RoboDK station: V1.rdk

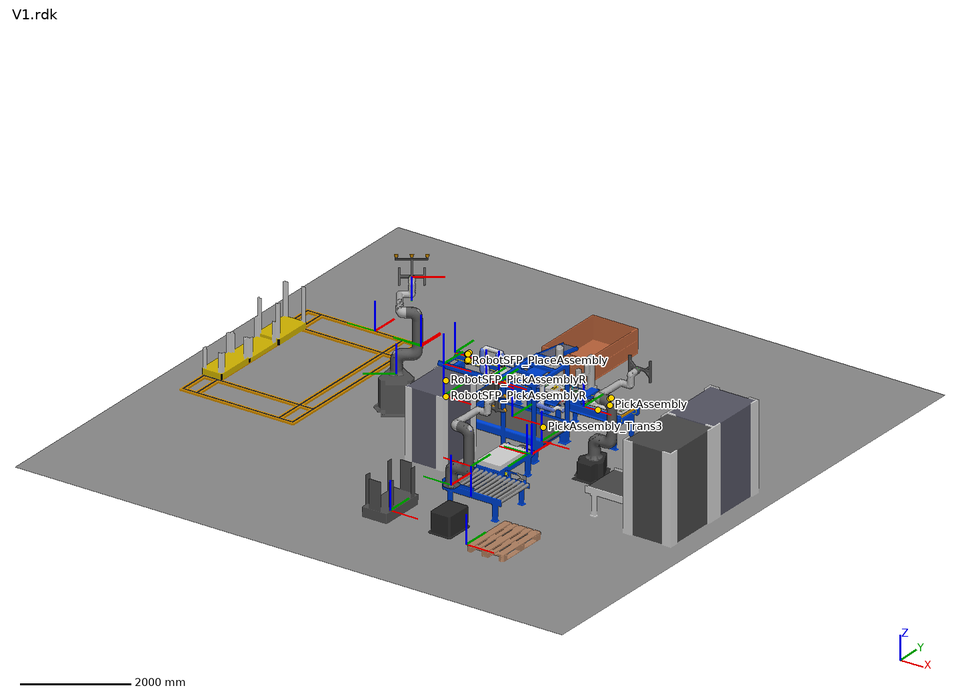
[picture v0: the station drawn from its stored meshes, robots at their saved joint values, targets as dots, program paths as lines]
Station V1 (saved by RoboDK 6.0.4). Poses are relative to the parent item; angles as X-Y-Z fixed-axis rotations.
Station parameters (name, value as stored): Assembly, 1, NextAssembly, 1, ScrewCircuit, 1, BuildCircuit, 1, UpFoamDone, 0, RackReady, 1, ActionGage_TwinTool, 0, TAGS, ['Assembly']
  - frame World at (0, 0, 0) mm
    - object Floor at (-130, -830, 0) mm, size 12000 x 12000 x 0 mm, geometry from UUID&
    - object Cell at (-1570, 1780, 20) mm, rotated rx 0 ry 0 rz 90 deg, size 7035 x 9205 x 1820 mm, geometry from UUID&
  - folder BaseAssembly Station
    - frame MainConveyor Base at (-1580, 450, 650) mm
      - robot MainConveyor: 1 axes
          modified DH rows (alpha deg, a mm, theta deg, d mm): 0, 0, 0, 0 linear
          base shift (0, 0, 0) mm, rotated rx 0 ry 90 rz 0 deg
          joint limits [-200000] to [200000]; home [0]; saved at [0]
        - frame MainConveyorRef at (90, -480, 0) mm
          - object TVAssemblies at (1835, 462, 0) mm, rotated rx 0 ry 0 rz -180 deg, size 1893 x 485 x 65 mm, geometry from UUID&
          - object AssemblyRack at (3909, 482, 2) mm, rotated rx 0 ry 0 rz 90 deg, size 40 x 853 x 485 mm, geometry from UUID&
          - object TVAssembly at (3594.88, 383.48, 47.7) mm, rotated rx 0 ry 0 rz 50 deg, size 853.3 x 900.2 x 46.5 mm, geometry from UUID&
      - frame DeltaRobot_Base at (1340, -530, 12) mm
        - frame Dobot Nova 5 Base at (-220, -80, 0) mm
          - robot Dobot Nova 5: 6 axes
              modified DH rows (alpha deg, a mm, theta deg, d mm): 0, 0, 0, 240; 90, 0, 90, 0; 0, 400, 0, 0; 0, 330, -90, 135; -90, 0, 0, 120; 90, 0, 180, 88
              joint limits [-360, -180, -160, -360, -360, -360] to [360, 180, 160, 360, 360, 360]; home [0, 0, -90, 0, 90, 0]; saved at [0, 0, -90, 0, 90, 0]
            - tool DeltaRobotTool, TCP at (0, 0, 130) mm, size 75 x 83 x 132.4 mm
          - object robot_support at (130, -180, 0) mm, size 257.4 x 257.4 x 15.4 mm, geometry from RoboDK-Logo-Plate-100x100mm.sld
      - frame MainConveyorRef_Init at (3165, -480, 0) mm
        - object TVAssemblies at (-1240, 462, 0) mm, rotated rx 0 ry 0 rz -180 deg, size 1893 x 485 x 65 mm, geometry from UUID&
        - object AssemblyRack at (834, 482, 2) mm, rotated rx 0 ry 0 rz 90 deg, size 40 x 853 x 485 mm, geometry from UUID&
        - object TVAssembly at (519.88, 383.48, 47.7) mm, rotated rx 0 ry 0 rz 50 deg, size 853.3 x 900.2 x 46.5 mm, geometry from UUID&
      - frame RobotSFP_Targets at (-1430, 980, -645) mm, rotated rx 0 ry 0 rz 90 deg
        - frame AssemblyRack_Targets at (0, 1000, 0) mm
          - target RobotSFP_PickAssemblyRack (Cartesian target) at (-2266, -3132, 478) mm, rotated rx 180 ry 0 rz -180 deg; joints [-130.241, 56.24, 97.421, -5.047, -77.391, -90.693] of Dobot CR30H
          - target RobotSFP_PickAssemblyRack_App (Cartesian target) at (-2266, -3132, 790) mm, rotated rx -180 ry 0 rz -180 deg; joints [-130.241, 25.611, 75.665, -5.962, -55.732, -88.432] of Dobot CR30H
          - target RobotSFP_PlaceAssemblyRack (Cartesian target) at (-1226, -2885, 690) mm, rotated rx 180 ry 0 rz -90 deg; joints [-92.609, 47.662, 66.312, -67.815, -58.973, -66.679] of Dobot CR30H
          - target RobotSFP_PlaceAssemblyRack_App (Cartesian target) at (-1226, -2885, 830) mm, rotated rx -180 ry 0 rz -90 deg; joints [-92.609, 38.532, 58.57, -72.434, -56.335, -58.059] of Dobot CR30H
        - frame TvAssembly at (0, 0, -20) mm
          - target RobotSFP_PlaceFrontPanel (Cartesian target) at (-1232.5, -1885.5, 730.48) mm, rotated rx 180 ry 0 rz -90 deg; joints [-92.924, 46.128, 65.422, -68.631, -58.762, -65.657] of Dobot CR30H
          - target RobotSFP_PlaceFrontPanel_App (Cartesian target) at (-1232.5, -1885.5, 863.5) mm, rotated rx -180 ry 0 rz -90 deg; joints [-92.924, 37.534, 57.905, -73.159, -56.297, -57.237] of Dobot CR30H
          - target RobotSFP_PlaceScreen (Cartesian target) at (-1189.8, -1890.5, 709.68) mm, rotated rx 180 ry 0 rz 90 deg; joints [-91.494, 45.247, 62.599, -68.849, -57.154, 117.178] of Dobot CR30H
          - target RobotSFP_PlaceScreen_App (Cartesian target) at (-1189.8, -1890.5, 871.7) mm, rotated rx 180 ry 0 rz 90 deg; joints [-91.494, 35.396, 53.282, -74.906, -54.246, 127.901] of Dobot CR30H
          - target RobotSFP_PlaceFrame (Cartesian target) at (-1219.5, -1885.2, 745.48) mm, rotated rx 180 ry 0 rz -90 deg; joints [-92.315, 45.44, 64.267, -68.683, -58.101, -64.505] of Dobot CR30H
          - target RobotSFP_PlaceFrame_App (Cartesian target) at (-1219.5, -1885.2, 853.5) mm, rotated rx -180 ry 0 rz -90 deg; joints [-92.315, 38.518, 58.189, -72.396, -56.073, -57.678] of Dobot CR30H
      - frame PickAssembly_Targets at (89.8, -480, -648) mm
        - target PickAssembly (Cartesian target) at (3485.2, 228, 693.7) mm, rotated rx -180 ry 0 rz -180 deg; joints [22.371, 48.063, -2.442, 0, 44.379, 112.371] of Dobot CR30H
        - target PickAssembly_App (Cartesian target) at (3485.2, 228, 823.7) mm, rotated rx -180 ry 0 rz -180 deg; joints [22.371, 43.327, -4.321, 0, 50.994, 112.371] of Dobot CR30H
        - target PickAssembly_Trans1 (Cartesian target) at (3525.2, 228, 853.7) mm, rotated rx 180 ry 5 rz 180 deg; joints [21.562, 41.902, -4.058, -5.74, 54.134, 115.007] of Dobot CR30H
        - target PickAssembly_Trans2 (Cartesian target) at (3605.2, -312, 853.7) mm, rotated rx -180 ry 0 rz 80 deg; joints [28.286, 14.78, 41.406, 0, 33.814, 218.286] of Dobot CR30H
        - target PickAssembly_Trans3 (Cartesian target) at (2776, -836.2, 483.7) mm, rotated rx -180 ry 0 rz 90 deg; joints [77.346, 50.715, 13.544, 0, 25.741, 257.346] of Dobot CR30H
    - frame Dobot CR30H Base at (-2010, -770, 600) mm, rotated rx 0 ry 0 rz 125 deg
      - robot Dobot CR30H: 6 axes
          modified DH rows (alpha deg, a mm, theta deg, d mm): 0, 0, 0, 386; 90, 0, 90, 0; 0, 840, 0, 0; 0, 740, -90, 277; -90, 0, 0, 220; 90, 0, 180, 211
          joint limits [-360, -360, -165, -360, -360, -360] to [360, 360, 165, 360, 360, 360]; home [0, 0, -90, 90, 90, 0]; saved at [0, 0, -90, 90, 90, 0]
        - frame ToolRobot1 Base at (0, 195, 425) mm, rotated rx -70 ry 0 rz 0 deg
          - robot ToolRobot1: 1 axes
              joint limits [-20] to [200]; home [0]; saved at [26]
        - tool ToolRobot1_TCP_Gripper, TCP at (0, 195, 425) mm, rotated rx -70 ry 0 rz 0 deg
        - tool ToolRobot1_TCP_Cup, TCP at (0, -240, 450) mm, rotated rx 70 ry 0 rz 0 deg
      - object Robot1_Stand at (0, 0, 0) mm, size 938.8 x 824.6 x 600 mm, geometry from UUID&
    - frame AssemblyRackConveyor Base at (1530, -1260, 440) mm
      - robot AssemblyRackConveyor: 1 axes
          modified DH rows (alpha deg, a mm, theta deg, d mm): 0, 0, 0, 0 linear
          base shift (0, 0, 0) mm, rotated rx 0 ry 90 rz 0 deg
          joint limits [-200000] to [200000]; home [0]; saved at [0]
        - frame AssemblyRackConveyorRef at (0, 0, 0) mm
      - frame AssemblyRackConveyorRef_Init at (0, 0, 0) mm
        - object AssemblyRack_Ref at (-1440, 0, 0) mm, size 40 x 853 x 485 mm, geometry from UUID&
        - object AssemblyRack_Ref at (-720, 0, 0) mm, size 40 x 853 x 485 mm, geometry from UUID&
        - object AssemblyRack_Ref at (-2160, 0, 0) mm, size 40 x 853 x 485 mm, geometry from UUID&
        - object AssemblyRack_Ref at (0, 0, 0) mm, size 40 x 853 x 485 mm, geometry from UUID&
  - folder Boxing Station
    - frame BoxingMachine Base at (1640, -1730, 385) mm, rotated rx 0 ry 0 rz 90 deg
      - robot BoxingMachine: 1 axes
          modified DH rows (alpha deg, a mm, theta deg, d mm): 0, 0, 0, 0 linear
          base shift (0, 0, 0) mm, rotated rx 0 ry 90 rz 0 deg
          joint limits [0] to [970]; home [0]; saved at [0]
        - frame BoxingMachine_Ref at (-150, 0, 60) mm, rotated rx 0 ry 0 rz 90 deg
          - object Foam at (255, 413.5, 93) mm, size 500 x 850 x 100 mm, geometry from UUID&
        - tool BoxingMachineTCP, TCP at (-650, 180, 120) mm
      - frame VaccumTool_Ref at (-1548.5, 251, 315) mm, rotated rx -180 ry 0 rz 90 deg
      - frame VaccumTool_Init at (-1548.5, 251, 315) mm, rotated rx -180 ry 0 rz 90 deg
        - object ClosedBox_Init at (-1, -21.5, 150) mm, rotated rx 180 ry 0 rz 180 deg, size 507 x 876.4 x 106.5 mm, geometry from UUID&
      - frame BoxingMachine_Init at (0, 0, 0) mm
        - object Foam_Ref at (-563.5, 255, 153) mm, rotated rx 0 ry 0 rz 90 deg, size 500 x 850 x 100 mm, geometry from UUID&
    - frame Pallet at (2510, -5020, 145) mm
      - object Pallet 1200mmx800mm 2 at (0, 0, 0) mm, size 800 x 1200 x 144.2 mm, geometry from UUID&
      - frame Pallet_Ref at (0, 0, 0) mm
    - frame Dobot CR30H Base at (1740, -4400, 870) mm, rotated rx 0 ry 0 rz 90 deg
      - robot Dobot CR30H: 6 axes
          modified DH rows (alpha deg, a mm, theta deg, d mm): 0, 0, 0, 386; 90, 0, 90, 0; 0, 840, 0, 0; 0, 740, -90, 277; -90, 0, 0, 220; 90, 0, 180, 211
          joint limits [-360, -360, -165, -360, -360, -360] to [360, 360, 165, 360, 360, 360]; home [0, 0, -90, 90, 90, 0]; saved at [0, 0, -90, 90, 90, 0]
        - tool VaccumTool, TCP at (0, 0, 150) mm, size 330 x 640 x 150 mm, geometry from VaccumTool.step
      - object RobotSTand at (-70, 0, -850) mm, size 660 x 500 x 420 mm, geometry from UUID&
    - frame OpenBoxDistributor at (420, -4430, 0) mm
      - object BoxDistributor at (0, 0, 0) mm, size 540 x 1000 x 800 mm, geometry from UUID&
      - frame OpenBoxDistributor_Ref at (0, 0, 0) mm
      - frame OpenBoxDistributor_Init at (0, 0, 0) mm
        - object OpenBox_Ref at (0, 0, 305) mm, size 506.5 x 962.1 x 106.4 mm, geometry from UUID&
        - object OpenBox_Ref at (0, 0, 411) mm, size 506.5 x 962.1 x 106.4 mm, geometry from UUID&
        - object OpenBox_Ref at (0, 0, 517) mm, size 506.5 x 962.1 x 106.4 mm, geometry from UUID&
        - object OpenBox_Ref at (0, 0, 623) mm, size 506.5 x 962.1 x 106.4 mm, geometry from UUID&
        - object OpenBox_Ref at (0, 0, 729) mm, size 506.5 x 962.1 x 106.4 mm, geometry from UUID&
        - object OpenBox_Ref at (0, 0, 835) mm, size 506.5 x 962.1 x 106.4 mm, geometry from UUID&
  - folder BackPanel Station
    - frame Dobot CR30H Base at (2580, -1120, 340) mm, rotated rx 0 ry 0 rz 90 deg
      - robot Dobot CR30H: 6 axes
          modified DH rows (alpha deg, a mm, theta deg, d mm): 0, 0, 0, 386; 90, 0, 90, 0; 0, 840, 0, 0; 0, 740, -90, 277; -90, 0, 0, 220; 90, 0, 180, 211
          joint limits [-360, -360, -165, -360, -360, -360] to [360, 360, 165, 360, 360, 360]; home [0, 0, -90, 90, 90, 0]; saved at [0, 0, -90, 90, 90, 0]
        - frame ToolRobot2 Base at (0, 0, 0) mm, rotated rx 180 ry 0 rz -90 deg
          - robot ToolRobot2: 1 axes
              joint limits [0] to [200]; home [0]; saved at [39]
      - object Robot1_Stand_S at (50, 0, 0) mm, size 751 x 659.7 x 336 mm, geometry from UUID&
    - frame PanelDistributor Base at (3400, -1180, 540) mm
      - robot PanelDistributor: 1 axes
          modified DH rows (alpha deg, a mm, theta deg, d mm): 0, 0, 0, 0 linear
          base shift (0, 0, 0) mm, rotated rx 0 ry 90 rz 0 deg
          joint limits [-200000] to [200000]; home [0]; saved at [-1400]
        - frame PanelDristributorRef at (0, 0, 0) mm
      - frame PanelDristributorRef_Init at (1400, 0, 0) mm
        - object TVBackPanel_Init at (220, 440, 30) mm, size 416 x 796.6 x 32 mm, geometry from UUID&
    - frame FoamDistributor Base at (3400, -2540, 540) mm
      - robot FoamDistributor: 1 axes
          modified DH rows (alpha deg, a mm, theta deg, d mm): 0, 0, 0, 0 linear
          base shift (0, 0, 0) mm, rotated rx 0 ry 90 rz 0 deg
          joint limits [-200000] to [200000]; home [0]; saved at [-1400]
        - frame FoamDristributorRef at (0, 0, 0) mm
      - frame FoamDristributorRef_Init at (1400, 0, 0) mm
        - object FoamDown_Init at (250, 430, 40) mm, size 500 x 850 x 50 mm, geometry from UUID&
        - object FoamTop_Init at (250, 430, 40) mm, size 500 x 850 x 50 mm, geometry from UUID&
  - folder ScrewCircuit Station
    - frame ScaraRobot1_Base at (1500, 220, 770) mm, rotated rx 0 ry 0 rz -90 deg
      - frame Dobot M1 Base at (-240, -190, -8) mm
        - robot Dobot M1: 4 axes, payload 1.5 kg, reach 446 mm, repeatability 0.01 mm, weight 14 kg
            modified DH rows (alpha deg, a mm, theta deg, d mm): 0, 0, 0, -53 linear; 0, 0, 0, 0; 0, 200, 0, 0; 180, 200, 0, 0
            joint limits [0, -90, -135, -180] to [250, 90, 135, 180]; home [200, -45, 90, 45]; saved at [250, -23.663, 76.911, 23.249]
          - tool Scara_ScrewDriverTool1 TCP, TCP at (0, 150, 205) mm
          - frame ScrewTool_AutoFeed Base at (0, 150, 205) mm
            - robot ScrewTool_AutoFeed1: 2 axes
                modified DH rows (alpha deg, a mm, theta deg, d mm): 0, 0, 0, 0 linear; 0, 0, 0, 0
                joint limits [-75, -200000] to [0, 200000]; home [0, 0]; saved at [-75, 0]
              - tool ScrewRefTcp1, TCP at (0, 0, 0) mm
              - frame ScrewRef1 at (0, 1000, 0) mm
            - frame ScrewRef_Init1 at (0, 0, -75) mm
              - object Screw_Ref at (0, 0, 6.5) mm, rotated rx -180 ry 0 rz 20 deg, size 5 x 4.9 x 7 mm, geometry from UUID&
        - object robot_support at (30, -130, -100) mm, size 257.4 x 257.4 x 15.4 mm, geometry from RoboDK-Logo-Plate-100x100mm.sld
    - frame ScaraRobot2_Base at (810, 220, 770) mm, rotated rx 0 ry 0 rz -90 deg
      - frame Dobot M1 Base at (-240, -190, -8) mm
        - robot Dobot M1: 4 axes, payload 1.5 kg, reach 446 mm, repeatability 0.01 mm, weight 14 kg
            modified DH rows (alpha deg, a mm, theta deg, d mm): 0, 0, 0, -53 linear; 0, 0, 0, 0; 0, 200, 0, 0; 180, 200, 0, 0
            joint limits [0, -90, -135, -180] to [250, 90, 135, 180]; home [200, -45, 90, 45]; saved at [200, -45, 90, 45]
          - tool Scara_ScrewDriverTool2 TCP, TCP at (0, 150, 205) mm
          - frame ScrewTool_AutoFeed Base at (0, 150, 205) mm
            - robot ScrewTool_AutoFeed2: 2 axes
                modified DH rows (alpha deg, a mm, theta deg, d mm): 0, 0, 0, 0 linear; 0, 0, 0, 0
                joint limits [-75, -200000] to [0, 200000]; home [0, 0]; saved at [-75, 0]
              - tool ScrewRefTcp2, TCP at (0, 0, 0) mm
              - frame ScrewRef2 at (0, 1000, 0) mm
            - frame ScrewRef_Init2 at (0, 0, -75) mm
              - object Screw_Ref at (0, 0, 6.5) mm, rotated rx -180 ry 0 rz 20 deg, size 5 x 4.9 x 7 mm, geometry from UUID&
        - object robot_support at (30, -130, -100) mm, size 257.4 x 257.4 x 15.4 mm, geometry from RoboDK-Logo-Plate-100x100mm.sld
  - folder InFeed Station
    - frame f_TV_Rack_Rail at (-3000, 1420, 0) mm, rotated rx 0 ry 0 rz 90 deg
      - robot m_TV_Rack_Panel: 2 axes
          modified DH rows (alpha deg, a mm, theta deg, d mm): 0, 0, 0, 0 linear; 90, 0, 0, 0 linear
          base shift (0, 0, 0) mm, rotated rx 0 ry 90 rz 0 deg
          joint limits [-3250, -2100] to [0, 0]; home [0, 0]; saved at [-710, -2100]
        - frame f_TV_Rack_Panel at (0, 0, 0) mm
        - tool t_TV_Rack_Panel, TCP at (0, 0, 200) mm
      - robot m_TV_Rack_Rim: 2 axes
          modified DH rows (alpha deg, a mm, theta deg, d mm): 0, 0, 0, 0 linear; 90, 0, 0, 0 linear
          base shift (0, 0, 0) mm, rotated rx 0 ry 90 rz 0 deg
          joint limits [-3250, -2100] to [0, 0]; home [0, 0]; saved at [-1600, -2100]
        - frame f_TV_Rack_Rim at (0, 0, 0) mm
        - tool t_TV_Rack_Rim, TCP at (0, 0, 200) mm
      - robot m_TV_Rack_Screen: 2 axes
          modified DH rows (alpha deg, a mm, theta deg, d mm): 0, 0, 0, 0 linear; 90, 0, 0, 0 linear
          base shift (0, 0, 0) mm, rotated rx 0 ry 90 rz 0 deg
          joint limits [-3250, -2100] to [0, 0]; home [0, 0]; saved at [-2480, -2100]
        - frame f_TV_Rack_Screen at (0, 0, 0) mm
        - tool t_TV_Rack_Screen, TCP at (0, 0, 200) mm
      - frame f_Ref_TV_Rack_Panel at (-1460, 2500, 0) mm, rotated rx 0 ry 0 rz 180 deg
        - object TVFrontPanel_Ref at (0, 0, 0) mm, size 812.6 x 460.3 x 32.5 mm, geometry from UUID&
        - object TVFrontPanel_Ref at (0, 0, 30) mm, size 812.6 x 460.3 x 32.5 mm, geometry from UUID&
        - object TVFrontPanel_Ref at (0, 0, 60) mm, size 812.6 x 460.3 x 32.5 mm, geometry from UUID&
        - object TVFrontPanel_Ref at (0, 0, 90) mm, size 812.6 x 460.3 x 32.5 mm, geometry from UUID&
        - object TVFrontPanel_Ref at (0, 0, 120) mm, size 812.6 x 460.3 x 32.5 mm, geometry from UUID&
        - object TVFrontPanel_Ref at (0, 0, 150) mm, size 812.6 x 460.3 x 32.5 mm, geometry from UUID&
        - object TVFrontPanel_Ref at (0, 0, 180) mm, size 812.6 x 460.3 x 32.5 mm, geometry from UUID&
        - object TVFrontPanel_Ref at (0, 0, 210) mm, size 812.6 x 460.3 x 32.5 mm, geometry from UUID&
        - object TVFrontPanel_Ref at (0, 0, 270) mm, size 812.6 x 460.3 x 32.5 mm, geometry from UUID&
        - object TVFrontPanel_Ref at (0, 0, 240) mm, size 812.6 x 460.3 x 32.5 mm, geometry from UUID&
        - object TVFrontPanel_Ref at (0, 0, 300) mm, size 812.6 x 460.3 x 32.5 mm, geometry from UUID&
        - object TVFrontPanel_Ref at (0, 0, 330) mm, size 812.6 x 460.3 x 32.5 mm, geometry from UUID&
        - object TVFrontPanel_Ref at (0, 0, 360) mm, size 812.6 x 460.3 x 32.5 mm, geometry from UUID&
        - object TVFrontPanel_Ref at (0, 0, 390) mm, size 812.6 x 460.3 x 32.5 mm, geometry from UUID&
        - object TVFrontPanel_Ref at (0, 0, 420) mm, size 812.6 x 460.3 x 32.5 mm, geometry from UUID&
        - object TVFrontPanel_Ref at (0, 0, 450) mm, size 812.6 x 460.3 x 32.5 mm, geometry from UUID&
      - frame f_Ref_TV_Rack_Rim at (-2350, 2500, 0) mm, rotated rx 0 ry 0 rz -180 deg
        - object TVRim_Ref at (0, 0, 0) mm, size 786.6 x 406 x 28 mm, geometry from UUID&
        - object TVRim_Ref at (0, 0, 15) mm, size 786.6 x 406 x 28 mm, geometry from UUID&
        - object TVRim_Ref at (0, 0, 30) mm, size 786.6 x 406 x 28 mm, geometry from UUID&
        - object TVRim_Ref at (0, 0, 45) mm, size 786.6 x 406 x 28 mm, geometry from UUID&
        - object TVRim_Ref at (0, 0, 60) mm, size 786.6 x 406 x 28 mm, geometry from UUID&
        - object TVRim_Ref at (0, 0, 75) mm, size 786.6 x 406 x 28 mm, geometry from UUID&
        - object TVRim_Ref at (0, 0, 90) mm, size 786.6 x 406 x 28 mm, geometry from UUID&
        - object TVRim_Ref at (0, 0, 105) mm, size 786.6 x 406 x 28 mm, geometry from UUID&
        - object TVRim_Ref at (0, 0, 120) mm, size 786.6 x 406 x 28 mm, geometry from UUID&
        - object TVRim_Ref at (0, 0, 135) mm, size 786.6 x 406 x 28 mm, geometry from UUID&
        - object TVRim_Ref at (0, 0, 225) mm, size 786.6 x 406 x 28 mm, geometry from UUID&
        - object TVRim_Ref at (0, 0, 210) mm, size 786.6 x 406 x 28 mm, geometry from UUID&
        - object TVRim_Ref at (0, 0, 195) mm, size 786.6 x 406 x 28 mm, geometry from UUID&
        - object TVRim_Ref at (0, 0, 180) mm, size 786.6 x 406 x 28 mm, geometry from UUID&
        - object TVRim_Ref at (0, 0, 165) mm, size 786.6 x 406 x 28 mm, geometry from UUID&
        - object TVRim_Ref at (0, 0, 150) mm, size 786.6 x 406 x 28 mm, geometry from UUID&
      - frame f_Ref_TV_Rack_Screen at (-2480, 2100, 0) mm
        - object TVScreen_Ref at (0, 0, 0) mm, size 776.6 x 396 x 12 mm, geometry from UUID&
        - object TVScreen_Ref at (0, 0, 12) mm, size 776.6 x 396 x 12 mm, geometry from UUID&
        - object TVScreen_Ref at (0, 0, 24) mm, size 776.6 x 396 x 12 mm, geometry from UUID&
        - object TVScreen_Ref at (0, 0, 36) mm, size 776.6 x 396 x 12 mm, geometry from UUID&
        - object TVScreen_Ref at (0, 0, 48) mm, size 776.6 x 396 x 12 mm, geometry from UUID&
        - object TVScreen_Ref at (0, 0, 60) mm, size 776.6 x 396 x 12 mm, geometry from UUID&
        - object TVScreen_Ref at (0, 0, 72) mm, size 776.6 x 396 x 12 mm, geometry from UUID&
        - object TVScreen_Ref at (0, 0, 84) mm, size 776.6 x 396 x 12 mm, geometry from UUID&
        - object TVScreen_Ref at (0, 0, 96) mm, size 776.6 x 396 x 12 mm, geometry from UUID&
        - object TVScreen_Ref at (0, 0, 108) mm, size 776.6 x 396 x 12 mm, geometry from UUID&
        - object TVScreen_Ref at (0, 0, 120) mm, size 776.6 x 396 x 12 mm, geometry from UUID&
        - object TVScreen_Ref at (0, 0, 132) mm, size 776.6 x 396 x 12 mm, geometry from UUID&
        - object TVScreen_Ref at (0, 0, 144) mm, size 776.6 x 396 x 12 mm, geometry from UUID&
        - object TVScreen_Ref at (0, 0, 180) mm, size 776.6 x 396 x 12 mm, geometry from UUID&
        - object TVScreen_Ref at (0, 0, 168) mm, size 776.6 x 396 x 12 mm, geometry from UUID&
        - object TVScreen_Ref at (0, 0, 156) mm, size 776.6 x 396 x 12 mm, geometry from UUID&
      - frame f_TV_Rack_Rail_Targets at (0, 0, 0) mm
        - target t_rack_panel_passive (joint target) at (-710, 2100, 200) mm; joints [-710, -2100] of m_TV_Rack_Panel
        - target t_rack_panel_lb (joint target) at (0, 2100, 200) mm; joints [0, -2100] of m_TV_Rack_Panel
        - target t_rack_panel_lt (joint target) at (0, 0, 200) mm; joints [0, 0] of m_TV_Rack_Panel
        - target t_rack_panel_active (joint target) at (-2480, 0, 200) mm; joints [-2480, 0] of m_TV_Rack_Panel
        - target t_rack_panel_rt (joint target) at (-3250, 0, 200) mm; joints [-3250, 0] of m_TV_Rack_Panel
        - target t_rack_panel_rb (joint target) at (-3250, 2100, 200) mm; joints [-3250, -2100] of m_TV_Rack_Panel
        - target t_rack_screen_passive (joint target) at (-2480, 2100, 200) mm; joints [-2480, -2100] of m_TV_Rack_Screen
        - target t_rack_screen_lb (joint target) at (0, 2100, 200) mm; joints [0, -2100] of m_TV_Rack_Screen
        - target t_rack_screen_lt (joint target) at (0, 0, 200) mm; joints [0, 0] of m_TV_Rack_Screen
        - target t_rack_screen_active (joint target) at (-710, 0, 200) mm; joints [-710, 0] of m_TV_Rack_Screen
        - target t_rack_screen_rt (joint target) at (-3250, 0, 200) mm; joints [-3250, 0] of m_TV_Rack_Screen
        - target t_rack_screen_rb (joint target) at (-3250, 2100, 200) mm; joints [-3250, -2100] of m_TV_Rack_Screen
        - target t_rack_rim_passive (joint target) at (-1600, 2100, 200) mm; joints [-1600, -2100] of m_TV_Rack_Rim
        - target t_rack_rim_lb (joint target) at (0, 2100, 200) mm; joints [0, -2100] of m_TV_Rack_Rim
        - target t_rack_rim_lt (joint target) at (0, 0, 200) mm; joints [0, 0] of m_TV_Rack_Rim
        - target t_rack_rim_active (joint target) at (-1600, 0, 200) mm; joints [-1600, 0] of m_TV_Rack_Rim
        - target t_rack_rim_rt (joint target) at (-3250, 0, 200) mm; joints [-3250, 0] of m_TV_Rack_Rim
        - target t_rack_rim_rb (joint target) at (-3250, 2100, 200) mm; joints [-3250, -2100] of m_TV_Rack_Rim
  - folder BackPanelScrew Station
    - frame RobotStandRef at (1230, -835, 20) mm
      - object Stand at (-145, 0, 0) mm, size 760 x 1160 x 1580 mm, geometry from UUID&
      - frame Dobot Nova 5 Base at (-90, 0, 1490) mm, rotated rx -180 ry 0 rz 0 deg
        - robot Dobot Nova 5: 6 axes
            modified DH rows (alpha deg, a mm, theta deg, d mm): 0, 0, 0, 240; 90, 0, 90, 0; 0, 400, 0, 0; 0, 330, -90, 135; -90, 0, 0, 120; 90, 0, 180, 88
            joint limits [-360, -180, -160, -360, -360, -360] to [360, 180, 160, 360, 360, 360]; home [0, 0, -90, 0, 90, 0]; saved at [0, 0, -90, 0, 90, 0]
          - frame ScrewTool_Panel Base at (62.5, 0, 70) mm, rotated rx 90 ry 0 rz 90 deg
            - robot ScrewTool_Panel: 2 axes
                modified DH rows (alpha deg, a mm, theta deg, d mm): 0, 0, 0, 0 linear; 0, 0, 0, 0
                joint limits [0, -200000] to [80, 200000]; home [0, 0]; saved at [0, 0]
              - frame BigScrewRef at (0, 0, 0) mm
            - frame BigScrewRef_Init at (0, 0, 70) mm, rotated rx -180 ry 0 rz 19.2 deg
              - object BigScrew_Ref at (0, 0, 0) mm, size 10 x 9.8 x 21 mm, geometry from UUID&
          - tool BigScrewRefTcp, TCP at (185, 0, 70) mm, rotated rx 0 ry 90 rz 0 deg
    - folder Python
      - Python program AutoScrewPanel (listed below)
      - Python program ResetAutoScrewPanel (listed below)
    - program AutoScrewP (4 instructions, listed below)
    - program ScrewPanelProcess (13 instructions, listed below)
  - folder CircuitAssembly Station
    - frame CircuitConveyor Base at (0, -190, 640) mm, rotated rx 0 ry 0 rz 90 deg
      - robot CircuitConveyorDoor: 1 axes
          modified DH rows (alpha deg, a mm, theta deg, d mm): 0, 0, 0, 0 linear
          joint limits [0] to [80]; home [0]; saved at [0]
      - robot CircuitConveyor: 1 axes
          modified DH rows (alpha deg, a mm, theta deg, d mm): 0, 0, 0, 0 linear
          base shift (0, 0, 0) mm, rotated rx 0 ry 90 rz 0 deg
          joint limits [-200000] to [200000]; home [0]; saved at [1430]
        - frame CircuitConveyorRef at (0, 10, 50) mm
      - frame CircuitConveyorRef_Init at (-1430, 10, 60) mm
        - object CircuitBox1 at (-80, 120, 15) mm, size 210 x 265 x 15 mm, geometry from UUID&
        - object Circuit1 at (-40, 170, 0) mm, size 158 x 88 x 12 mm, geometry from UUID&
        - object Circuit2 at (-60, 80, 20) mm, size 113 x 88 x 12 mm, geometry from UUID&
        - object Circuit3 at (-60, 220, 0) mm, size 58 x 38 x 4 mm, geometry from UUID&
        - object Circuit4 at (-50, 60, 0) mm, size 148 x 88 x 9 mm, geometry from UUID&
        - object Circuit5 at (-60, 190, 20) mm, size 106 x 63 x 13 mm, geometry from UUID&
        - object Circuit6 at (-170, 130, 20) mm, size 12 x 232 x 5 mm, geometry from UUID&
        - object Circuit7 at (-170, 120, 0) mm, size 28 x 258 x 6 mm, geometry from UUID&
        - object CircuitBox2 at (-80, 120, 30) mm, size 210 x 265 x 15 mm, geometry from UUID&
    - frame RollerConveyor Base at (10, 1990, 560) mm, rotated rx 0 ry 0 rz 90 deg
      - object Container at (-190, -370, -560) mm, rotated rx 0 ry 0 rz -90 deg, size 1000 x 1600 x 500 mm, geometry from UUID&
      - robot RollerConveyor: 1 axes
          modified DH rows (alpha deg, a mm, theta deg, d mm): 0, 0, 0, 0 linear
          base shift (0, 0, 0) mm, rotated rx 180 ry 82.41 rz 180 deg
          joint limits [-20000] to [20000]; home [0]; saved at [0]
        - frame RollerConveyorRef at (0, 0, 0) mm
      - object CircuitBox2 at (280, 0, -520) mm, rotated rx 0 ry 0 rz -45 deg, size 210 x 265 x 15 mm, geometry from UUID&
      - object CircuitBox1 at (390, 340, -520) mm, rotated rx 0 ry 0 rz 25 deg, size 210 x 265 x 15 mm, geometry from UUID&
  - Python program main (listed below)

--- Python program AutoScrewPanel ---
# Type help("robodk.robolink") or help("robodk.robomath") for more information
# Press F5 to run the script
# Documentation: https://robodk.com/doc/en/RoboDK-API.html
# Reference:     https://robodk.com/doc/en/PythonAPI/robodk.html
# Note: It is not required to keep a copy of this file, your Python script is saved with your RDK project

# You can also use the new version of the API:
from robodk import robolink    # RoboDK API
from robodk import robomath    # Robot toolbox
RDK = robolink.Robolink()

# Forward and backwards compatible use of the RoboDK API:
# Remove these 2 lines to follow python programming guidelines
from robodk import *      # RoboDK API
from robolink import *    # Robot toolbox
# Link to RoboDK
# RDK = Robolink()
# Type help("robolink") or help("robodk") for more information
# Press F5 to run the script
# Documentation: https://robodk.com/doc/en/RoboDK-API.html
# Reference:     https://robodk.com/doc/en/PythonAPI/index.html
# Note: It is not required to keep a copy of this file, your python script is saved with the station



#----- Constante -----
NEW_REF_OBJECT_NAME = 'BigScrew_Ref' #Name of the ref object to copy
NEW_OBJECT_NAME = 'BigScrew' #Name of the new object created
REFERENCE_FRAME = 'BigScrewRef' #Name of the frame the object will move to
REFERENCE_FRAME_REF = 'BigScrewRef_Init'
MECHANISM_NAME = 'ScrewTool_Panel'
PART_TRAVEL_MM = 75 #Travel for each panel

mechanism = RDK.Item(MECHANISM_NAME,itemtype=robolink.ITEM_TYPE_ROBOT)

#------- Program ------
frame = RDK.Item(REFERENCE_FRAME, robolink.ITEM_TYPE_FRAME)
frame_ref = RDK.Item(REFERENCE_FRAME_REF, robolink.ITEM_TYPE_FRAME)
ref_obj = RDK.Item(NEW_REF_OBJECT_NAME, robolink.ITEM_TYPE_OBJECT)


RDK.Render(False)

if mechanism.Valid():
    mechanism.setJoints([0,0])

if frame.Valid():
    for item in frame.Childs():
        if item.Type() == robolink.ITEM_TYPE_OBJECT:
            item.Delete()



for item in frame_ref.Childs():
    if frame.Valid() and  ref_obj.Valid():
        item.Copy()
        new_obj = RDK.Paste()
        new_obj.setVisible(False)
        new_obj.setParent(frame_ref)
        new_obj.setName(NEW_OBJECT_NAME)
        RDK.Update()
        new_obj.setParentStatic(frame)
        new_obj.setVisible(True)
RDK.Render(True)


if mechanism.Valid():
    mechanism.MoveJ([70,800])

--- Python program ResetAutoScrewPanel ---
# Type help("robodk.robolink") or help("robodk.robomath") for more information
# Press F5 to run the script
# Documentation: https://robodk.com/doc/en/RoboDK-API.html
# Reference:     https://robodk.com/doc/en/PythonAPI/robodk.html
# Note: It is not required to keep a copy of this file, your Python script is saved with your RDK project

# You can also use the new version of the API:
from robodk import robolink    # RoboDK API
from robodk import robomath    # Robot toolbox
RDK = robolink.Robolink()

# Forward and backwards compatible use of the RoboDK API:
# Remove these 2 lines to follow python programming guidelines
from robodk import *      # RoboDK API
from robolink import *    # Robot toolbox
# Link to RoboDK
# RDK = Robolink()
# Type help("robolink") or help("robodk") for more information
# Press F5 to run the script
# Documentation: https://robodk.com/doc/en/RoboDK-API.html
# Reference:     https://robodk.com/doc/en/PythonAPI/index.html
# Note: It is not required to keep a copy of this file, your python script is saved with the station



#----- Constante -----
NEW_REF_OBJECT_NAME = 'BigScrew_Ref' #Name of the ref object to copy
NEW_OBJECT_NAME = 'BigScrew' #Name of the new object created
REFERENCE_FRAME = 'BigScrewRef' #Name of the frame the object will move to
REFERENCE_FRAME_REF = 'BigScrewRef_Init'
MECHANISM_NAME = 'ScrewTool_Panel'
PART_TRAVEL_MM = 75 #Travel for each panel


mechanism = RDK.Item(MECHANISM_NAME,itemtype=robolink.ITEM_TYPE_ROBOT)

#------- Program ------
frame = RDK.Item(REFERENCE_FRAME, robolink.ITEM_TYPE_FRAME)
frame_ref = RDK.Item(REFERENCE_FRAME_REF, robolink.ITEM_TYPE_FRAME)
ref_obj = RDK.Item(NEW_REF_OBJECT_NAME, robolink.ITEM_TYPE_OBJECT)


RDK.Render(False)



if frame.Valid():
    for item in frame.Childs():
        if item.Type() == robolink.ITEM_TYPE_OBJECT:
            item.Delete()

RDK.Render(True)


if mechanism.Valid():
    mechanism.MoveJ([0,800])

if mechanism.Valid():
    mechanism.setJoints([0,0])

--- program AutoScrewP (robot Dobot M1) ---
  Call AutoScrewPanel
  Attach to BigScrewRefTcp
  Detach from BigScrewRefTcp
  Call ResetAutoScrewPanel

--- program ScrewPanelProcess (robot Dobot Nova 5) ---
  Set Ref.: BackPanelScrew_Targets at (90, 0, 1150) mm, rotated rx 180 ry 0 rz 0 deg
  Set Tool: BigScrewRefTcp
  MoveJ (BackPanelScrew_Home) [its target is no longer in the station]
  MoveJ (BackPanelScrew_Target1) [its target is no longer in the station]
  Call AutoScrewP
  MoveL (BackPanelScrew_Target2) [its target is no longer in the station]
  Call AutoScrewP
  MoveL (BackPanelScrew_Target3) [its target is no longer in the station]
  Call AutoScrewP
  MoveL (BackPanelScrew_Target4) [its target is no longer in the station]
  Call AutoScrewP
  MoveJ (BackPanelScrew_Home) [its target is no longer in the station]
  Call PickTv

--- Python program main ---
import sys

sys.path.append(
    r'P:\Robodk Codesys Intergration\bridge\.venv\Lib\site-packages')
sys.path.append(r'P:\Robodk Codesys Intergration\bridge')


if __name__ == '__main__':
    from bridge.rdk import main

    main()
